// TIA Portal V21 export
VAR_GLOBAL   // PLC tag table "K_Zona_Sterilizzatore"
END_VAR
